{attribute 'GeneratedUsingTerminal: EK1100-0000-0018'}
{attribute addProperty BoxType "EK1100-0000-0018"}
{attribute addProperty Id "Beckhoff_EKx9xxEK1122Beckhoff_EKx9xxEK1122_4392AD201154"}
{attribute addProperty CRC "2523386168"}
{attribute addProperty Size "1154"}
TYPE Beckhoff_EKx9xx_9667D138 EXTENDS EK1100_AB5A9467 :
STRUCT
	{attribute addProperty Name "Beckhoff_EKx9xxEK1122"}
	{attribute addProperty PreviousPort "Beckhoff EKx9xx : B"}
	Beckhoff_EKx9xxEK1122 : Beckhoff_EKx9xxEK1122_4392AD20;
END_STRUCT
END_TYPE

(* stored: Version 1.2.0.0, ProductVersion 3.1.4024.9
   DUT Beckhoff_EKx9xx_9667D138: Id {422ac62d-57da-46e9-962b-f1579b64106d} *)
